(* CODESYS project GVL_AXIS_GROUP.gvl.xml

Project tree, tasks and I/O mapping:
  global variables GVL_AXIS_GROUP
*)

// GVL_AXIS_GROUP
{attribute 'qualified_only'}
VAR_GLOBAL
	AxisGroup : ST_AXIS_GROUP; // Команды, статусы и диагностика группы XYZ
END_VAR
